KUKA KRL program: hp023.src, hp023.dat

--- hp023.src ---
&ACCESS RVP
&REL 1
&COMMENT ATEGO STB
&PARAM DISKPATH = KRC:\R1\Program
&PARAM TEMPLATE = C:\KRC\Roboter\Template\vorgabe
&PARAM EDITMASK = *
DEF hp023( )
;FOLD INI
  ;FOLD BASISTECH INI
    GLOBAL INTERRUPT DECL 3 WHEN $STOPMESS==TRUE DO IR_STOPM ( )
    INTERRUPT ON 3
    BAS (#INITMOV,0)
  ;ENDFOLD (BASISTECH INI)
;FOLD GRIPPERTECH INI
USER_GRP(0,DUMMY,DUMMY,GDEFAULT)
;ENDFOLD (GRIPPERTECH INI)
  ;FOLD USER INI
    ;Make your modifications here

  ;ENDFOLD (USER INI)
     ;FOLD COLLISION_V_3.01 INI ;%{E}
        IF (COLLISION_DATA[1].I_NR>0) THEN
          GLOBAL INTERRUPT DECL 21 WHEN $IN[COLLISION_DATA[1].I_NR]==FALSE DO COLLSTOP (1,0 )
        ENDIF
        IF (COLLISION_DATA[2].I_NR>0) THEN
          GLOBAL INTERRUPT DECL 22 WHEN $IN[COLLISION_DATA[2].I_NR]==FALSE DO COLLSTOP (2,0 )
        ENDIF
        IF (COLLISION_DATA[3].I_NR>0) THEN
          GLOBAL INTERRUPT DECL 23 WHEN $IN[COLLISION_DATA[3].I_NR]==FALSE DO COLLSTOP (3,0 )
        ENDIF
        IF (COLLISION_DATA[4].I_NR>0) THEN
          GLOBAL INTERRUPT DECL 24 WHEN $IN[COLLISION_DATA[4].I_NR]==FALSE DO COLLSTOP (4,0 )
        ENDIF
     ;ENDFOLD (COLLISION)
;ENDFOLD (INI)

; Caracterização dos meios de produção
; Changes: HP023 - Atego STB
; Versão Atual: 28/03/2016
; Name: P13.050-R1

chk_w8_wechs_ok ( )         ; CHECK TOOL CHANGE

MBINI( )                    ; RESET SINAIS

$TIMER[8]=0
$TIMER_STOP[8]=FALSE

;FOLD PTP HOME  Vel=100 % DEFAULT;%{PE}%MKUKATPBASIS,%CMOVE,%VPTP,%P 1:PTP, 2:HOME, 3:, 5:100, 7:DEFAULT
$BWDSTART = FALSE
PDAT_ACT=PDEFAULT
FDAT_ACT=FHOME
BAS(#PTP_PARAMS,100)
$H_POS=XHOME
PTP XHOME
;ENDFOLD

WKZ11_AN ( )                ; Pega Gripper 913

HO_COM_03_AG01_G02 ( )      ; Pega Traseira

AB_COM_03_ST01_G02 ( )      ; Deposita Traseira

WKZ4_AN ( )                 ; Pega Gun C3

PS_A_STB_GEO_C03 ( )        ; Solda Geometria

WKZ4_AB ( )                 ; Deposita Gun C3

WKZ11_ETB_STB_OFF( )        ; Pega Gripper GeoBox

WKZ11_AB ( )                ; Deposita Gripper 913

WKZ4_AN ( )                 ; Pega Gun C3

;FOLD ; ;%{PE}%R 8.2.20,%MKUKATPBASIS,%CCOMMENT,%VNORMAL,%P 2:
;ENDFOLD
PS_A_STB_RES_C03 ( )        ; Solda Respot

WKZ4_AB ( )                 ; Deposita Gun C3

;FOLD PTP HOME  Vel=100 % DEFAULT;%{PE}%MKUKATPBASIS,%CMOVE,%VPTP,%P 1:PTP, 2:HOME, 3:, 5:100, 7:DEFAULT
$BWDSTART = FALSE
PDAT_ACT=PDEFAULT
FDAT_ACT=FHOME
BAS(#PTP_PARAMS,100)
$H_POS=XHOME
PTP XHOME
;ENDFOLD

$TIMER_STOP[8]=TRUE

END

--- hp023.dat ---
&ACCESS RVP
&REL 1
&COMMENT ATEGO STB
&PARAM DISKPATH = KRC:\R1\Program
&PARAM TEMPLATE = C:\KRC\Roboter\Template\vorgabe
&PARAM EDITMASK = *
DEFDAT hp023
;FOLD EXTERNAL DECLARATIONS;%{PE}%MKUKATPBASIS,%CEXT,%VCOMMON,%P
;FOLD GRIPPERTECH EXT
EXT  H50 (INT  :IN,INT  :IN,INT  :IN,GRP_TYP  :IN )
;ENDFOLD (GRIPPERTECH EXT)
;FOLD SPOTTECH EXT
EXT  USERSPOT (S_COMMAND  :IN,SPOT_TYPE  :IN )
;ENDFOLD (SPOTTECH EXT)
;FOLD BASISTECH EXT;%{PE}%MKUKATPBASIS,%CEXT,%VEXT,%P
EXT  BAS (BAS_COMMAND  :IN,REAL  :IN )
DECL INT SUCCESS
;ENDFOLD (BASISTECH EXT)
;FOLD USER EXT;%{E}%MKUKATPUSER,%CEXT,%VEXT,%P
;Make your modifications here

;ENDFOLD (USER EXT)
;ENDFOLD (EXTERNAL DECLARATIONS)
DECL SPOT_SUGG_T LAST_SPOT={GUN[] " 1                      ",RETR_CMD[] "#OPN                    ",CHOISE[] "#FIRST                  ",CLO_TM[] "0                       ",PGNO1[] " 1                      ",PRESS1[] "0                       ",PGNO2[] " 1                      ",PRESS2[] "0                       ",SPOT_PARAMS[] "NORMAL                  "}
DECL BASIS_SUGG_T LAST_BASIS={POINT1[] "PS01010001              ",POINT2[] "PS01010001              ",CP_PARAMS[] "CPDAT0                  ",PTP_PARAMS[] "PDAT0                   ",CONT[] "                        ",CP_VEL[] "2                       ",PTP_VEL[] " 100                    ",SPL_NAME[] "S0                      "}
ENDDAT
